Staubli VAL3: tool.dtx

num nIndex
num nIndexTool
num nKey
public num nPage
num nRefresh
num nTime = 1
num nView
string sEvent
public string sItems
string sList
string sMenu
string sMessage
string sMenu8[8]
string sActionON[3]
string sActionOFF[3]
bool bButton[8]
bool bLarge
InstrItem iInstrTcpON[3]
  [0]
    string sType
    string sData
  [1]
    string sType
    string sData
  [2]
    string sType
    string sData
InstrItem iInstrTcpOFF[3]
  [0]
    string sType
    string sData
  [1]
    string sType
    string sData
  [2]
    string sType
    string sData
tool tTool = {fatherId=flange[0], ioLink=valve1}
string sSession
frame fFrame = {fatherId=world[0]}
